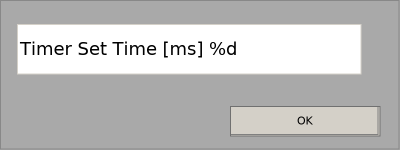
VISUALIZATION DialogTimer_GripperOpenClose  // 400x150
    Button (230,106 150x30), "OK"
        OnMouseClick: CloseDialog Dialog=DialogTimer_GripperOpenClose, Result=OK, NumpadKeypadSet=True
    Textfield (17,24 344x50), "Timer Set Time [ms] %d", text variable: PersistentStruct.TimeGripperOpen
        OnMouseClick: write the text variable via Edit
END_VISUALIZATION

(* stored: Version 1.1.0.1, ProductVersion 3.1.4024.3
   Visu DialogTimer_GripperOpenClose: Id {30a53c75-9193-466d-b3bb-7896636af38c} *)
